# EPICS substitutions: src/makeBaseApp/top/pcdsIocBoot/ioc/_IOC_.substitutions
# IOC archive file
## Replace _IOCPVROOT_ with the PV prefix used for
## iocAdmin PV's on this IOC

# Generate IOC archive request
file archive__APPNAME_.archive
{
	{ IOC = "_IOCPVROOT_" }
}
